FUNCTION_BLOCK FB_StateOpening
VAR_IN_OUT
	stAxis  	: ARRAY [GVL.cXP .. GVL.cXM] OF ST_AxisGroup;	
	bTopEntry	: BOOL;
END_VAR
VAR_INPUT
	nRet	: INT;
	fSpeed	: LREAL;
END_VAR
VAR_OUTPUT
	bBusy	: BOOL;
END_VAR
VAR
	//state-machine
	nCurrentState	: INT;
	nNextState		: INT;
	
END_VAR

//////////////////////////////////////////////////
//Puts shutter in open position					//
//////////////////////////////////////////////////
IF bTopEntry = TRUE THEN
	bTopEntry 	:= FALSE;
	nNextState 	:= 1100;
END_IF
bBusy 	:= TRUE;
nCurrentState 	:= nNextState;

CASE nCurrentState OF
(*Perform Open Shutter Motion*)
	1100:
		IF nRet = GVL.cXP THEN
			stAxis[GVL.cXP].mcMoveAbs(Axis:=stAxis[GVL.cXP].axisRef, Position:=GVL.cPosStart, Velocity:=fSpeed, Execute:=TRUE);
		ELSIF nRet = GVL.cXM THEN	
			stAxis[GVL.cXM].mcMoveAbs(Axis:=stAxis[GVL.cXM].axisRef, Position:=GVL.cPosEnd, Velocity:=fSpeed, Execute:=TRUE);
		END_IF
		IF stAxis[GVL.cXP].mcMoveAbs.Done OR stAxis[GVL.cXM].mcMoveAbs.Done THEN
			stAxis[GVL.cXP].mcMoveAbs(Axis:=stAxis[GVL.cXP].axisRef, Execute:=FALSE);
			stAxis[GVL.cXM].mcMoveAbs(Axis:=stAxis[GVL.cXM].axisRef, Execute:=FALSE);
			nNextState := 1110;
		END_IF	
		
	1110: //End action
		bBusy := FALSE;

END_CASE

END_FUNCTION_BLOCK

(* stored: Version 1.1.0.1, ProductVersion 3.1.4020.12
   POU FB_StateOpening: Id {fa4bcf8d-b0de-4a28-a87c-d71c04474993}, SpecialFunc None *)
